FUNCTION_BLOCK FB_SystemTime
VAR_INPUT
END_VAR
VAR_OUTPUT
END_VAR
VAR
	GetLocalSystemTime 	: FB_LocalSystemTime;
	wDateW				: WORD;
END_VAR

GetLocalSystemTime(bEnable := TRUE);

PROPERTY dtDateTimeFull : DT
GET
dtDateTimeFull 	:= SYSTEMTIME_TO_DT(GetLocalSystemTime.systemTime);
END_GET
END_PROPERTY

PROPERTY sDate : STRING
GET
sDate	:= MID(sDateTimeFull,10,1);
END_GET
END_PROPERTY

PROPERTY sDateTime : STRING
GET
sDateTime := MID(sDateTimeFull,19,1);
END_GET
END_PROPERTY

PROPERTY sDateTimeFull : STRING
GET
sDateTimeFull 	:= SYSTEMTIME_TO_STRING(GetLocalSystemTime.systemTime);
END_GET
END_PROPERTY

PROPERTY sDayOfWeek : STRING
GET
wDateW	:=  GetLocalSystemTime.systemTime.wDayOfWeek;
IF wDateW = 0 THEN
	sDayOfWeek := 'Sunday';
ELSIF wDateW = 1 THEN
	sDayOfWeek := 'Monday';
ELSIF wDateW = 2 THEN
	sDayOfWeek := 'Tuesday';
ELSIF wDateW = 3 THEN
	sDayOfWeek := 'Wednesday';
ELSIF wDateW = 4 THEN
	sDayOfWeek := 'Thursday';
ELSIF wDateW = 5 THEN
	sDayOfWeek := 'Friday';
ELSIF wDateW = 6 THEN
	sDayOfWeek := 'Saturday';
END_IF
END_GET
END_PROPERTY

PROPERTY sTime : STRING
GET
sTime := MID(sDateTimeFull,8,12);
END_GET
END_PROPERTY

PROPERTY wDay : Word
GET
wDay :=  GetLocalSystemTime.systemTime.wDay;
END_GET
END_PROPERTY

PROPERTY wHour : WORD
GET
wHour	:=	GetLocalSystemTime.systemTime.wHour;
END_GET
END_PROPERTY

PROPERTY wMilliSeconds : WORD
GET
wMilliseconds	:=	GetLocalSystemTime.systemTime.wMilliseconds;
END_GET
END_PROPERTY

PROPERTY wMinute : WORD
GET
wMinute	:=	GetLocalSystemTime.systemTime.wMinute;
END_GET
END_PROPERTY

PROPERTY wMonth : Word
GET
wMonth	:=  GetLocalSystemTime.systemTime.wMonth;
END_GET
END_PROPERTY

PROPERTY wSecond : WORD
GET
wSecond	:=	GetLocalSystemTime.systemTime.wSecond;
END_GET
END_PROPERTY

PROPERTY wYear : Word
GET
wYear :=  GetLocalSystemTime.systemTime.wYear;
END_GET
END_PROPERTY

END_FUNCTION_BLOCK

(* stored: Version 1.1.0.1, ProductVersion 3.1.4024.12
   POU FB_SystemTime: Id {31552c93-32b7-4f00-a134-e901f8c7c218}, SpecialFunc None
   Property dtDateTimeFull: Id {d55bf6a2-5378-4d0d-bd4a-5f9d6788fe6c}
   Get Get: Id {5e41d91a-f35f-4a42-96f5-52d39bfa7541}
   Property sDate: Id {1c599e7c-ea74-4cd5-978a-1ec2ddb7ed4c}
   Get Get: Id {0956643a-df73-40c8-94a2-7d324c3465fe}
   Property sDateTime: Id {03f9a243-6aea-4a60-955e-ac73c22ea7e8}
   Get Get: Id {7f508d2c-8cde-48e5-9448-df7f5c8d5945}
   Property sDateTimeFull: Id {bd750e46-94af-4a5c-9fa8-045960809265}
   Get Get: Id {60f2610d-ab67-4424-bf59-3114699a0b73}
   Property sDayOfWeek: Id {fc363c62-735b-4c86-a93f-1f2138738875}
   Get Get: Id {25e5ed67-b5ca-4b1c-aff9-6fffcb20b5cc}
   Property sTime: Id {4fe46746-6e68-4dd1-930f-748eaea121ea}
   Get Get: Id {59f93972-8a88-4464-99c6-21ad1926dff1}
   Property wDay: Id {286f771c-0932-4030-bf78-bcb551a2b48e}
   Get Get: Id {4ba9387f-472e-48e5-9fcb-d00f48840d88}
   Property wHour: Id {a4f3c154-2011-43b4-a917-80acff9d0ab3}
   Get Get: Id {957542ff-0af3-4de5-8b9b-10e27bdb7b11}
   Property wMilliSeconds: Id {179e4f99-e501-41dd-b893-b4b386b545c4}
   Get Get: Id {9659eab7-1049-4d15-9b03-1ef716fd347d}
   Property wMinute: Id {7628e342-7dc7-45cb-abae-e59d54e08b33}
   Get Get: Id {407a1750-eeea-4f93-889b-d1b297721062}
   Property wMonth: Id {3319d4ec-f4d3-40ca-b2e3-cc7bdb570352}
   Get Get: Id {d6d1debe-40ad-4854-be42-bbe5004ae68a}
   Property wSecond: Id {7fc37835-33d7-4beb-9c8c-f2a2158b0cba}
   Get Get: Id {1046b553-d70d-4091-9bc3-178e237491f0}
   Property wYear: Id {0228e2b4-a364-46e1-8420-7b6362967808}
   Get Get: Id {401493e0-fb57-40c3-9e55-194f2355520c} *)
